// SIMATIC STEP 7 (V5.x) project TIAWinAC
// CPU: PLCSim
// station: P_ADR_BUS
// station: Configuration
// station: SoftPLC
// program: WinAC

SYMBOL_TABLE
"Example variables"	FB 1	FB 1
"MW10Counter"	M 0.0	BOOL	// 0=No addition, 1=Add 1 to previous count in MW10 each scan
"MW12Counter"	M 0.1	BOOL	// 0=No subtraction, 1=Subtract 2 from previous count in MW12 each scan
"MW14Counter"	M 0.2	BOOL	// 0=No addition, 1=Add 3 to previous count in MW14 each scan
"MW10"	MW 10	INT	// The sum of the number of scans
"MW12"	MW 12	INT	// The differnce of the number of scans decremented by twos
"MW14"	MW 14	INT	// The sum of the number of scans incremented by 3
"WinCC Lab 2"	VAT 1	
END_SYMBOL_TABLE

FUNCTION_BLOCK "Example variables"	// FB 1
VERSION : 0.1
VAR_INPUT
  One : INT ;
END_VAR
VAR_OUTPUT
  Two : INT ;
END_VAR
VAR
  Three : INT ;
END_VAR
VAR_TEMP
  Four : INT ;
END_VAR
BEGIN
NETWORK
TITLE =
END_FUNCTION_BLOCK

DATA_BLOCK DB 1
VERSION : 0.0
"Example variables"
BEGIN
END_DATA_BLOCK

ORGANIZATION_BLOCK OB 1
TITLE = "Main Program Sweep (Cycle)"
//WinLC Program for use in the WinCC Configuration course.
//
//Logic in this block will be executed every scan.
VERSION : 0.1
VAR_TEMP
  OB1_EV_CLASS : BYTE ;	//Bits 0-3 = 1 (Coming event), Bits 4-7 = 1 (Event class 1)
  OB1_SCAN_1 : BYTE ;	//1 (Cold restart scan 1 of OB 1), 3 (Scan 2-n of OB 1)
  OB1_PRIORITY : BYTE ;	//1 (Priority of 1 is lowest)
  OB1_OB_NUMBR : BYTE ;	//1 (Organization block 1, OB1)
  OB1_RESERVED_1 : BYTE ;	//Reserved for system
  OB1_RESERVED_2 : BYTE ;	//Reserved for system
  OB1_PREV_CYCLE : INT ;	//Cycle time of previous OB1 scan (milliseconds)
  OB1_MIN_CYCLE : INT ;	//Minimum cycle time of OB1 (milliseconds)
  OB1_MAX_CYCLE : INT ;	//Maximum cycle time of OB1 (milliseconds)
  OB1_DATE_TIME : DATE_AND_TIME ;	//Date and time OB1 started
  Output : INT ;
END_VAR
BEGIN
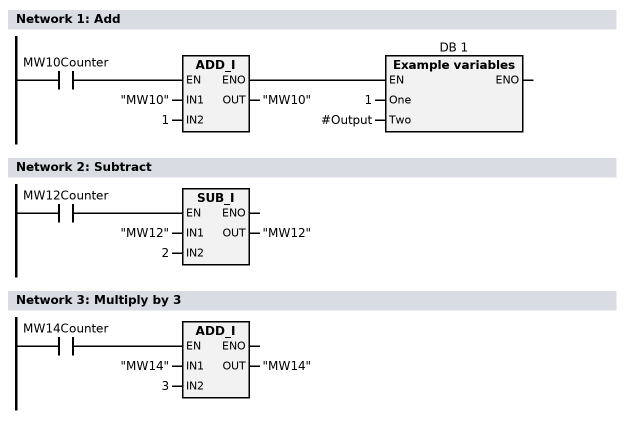
NETWORK
TITLE = Add
//When bit M0.0 = 1 then increment MW10 by 1 each scan, when M0.0 = 0 do no 
//addition, just retain the previous sum.
      A(;
      A     "MW10Counter";
      JNB   _001;
      L     "MW10";
      L     1;
      +I;
      T     "MW10";
      AN    OV;
      SAVE;
      CLR;
_001: A     BR;
      );
      JNB   _004;
      CALL  "Example variables" , DB 1 (
           One                      := 1,
           Two                      := #Output);
_004: NOP   0;
NETWORK
TITLE = Subtract
//When bit M0.1 = 1 then decrement MW12 by 2 each scan, when M0.1 = 0 do no 
//subtraction, just retain the previous difference.
      A     "MW12Counter";
      JNB   _005;
      L     "MW12";
      L     2;
      -I;
      T     "MW12";
_005: NOP   0;
NETWORK
TITLE = Multiply by 3
//When bit M0.2 = 1 then increment MW14 by 3 each scan, when M0.2 = 0 do no 
//addition, just retain the previous sum.
      A     "MW14Counter";
      JNB   _006;
      L     "MW14";
      L     3;
      +I;
      T     "MW14";
_006: NOP   0;
END_ORGANIZATION_BLOCK
